{attribute 'qualified_only'}
VAR_GLOBAL
	MasterStopPB_Pressed		: BOOL;
	CageEstopCircuitOK			: BOOL;
	RemoteModeSelected			: BOOL;
	PSU1_DCOK					: BOOL;
END_VAR

(* stored: Version 1.1.0.1, ProductVersion 3.1.4024.11
   GVL MCP_IO: Id {2eccccd0-d6b2-453f-b49b-33f7d0364904} *)
